PROGRAM Manual_1
VAR
	running: BOOL;
	currentError: UDINT;
	manualMode: E_JogMode;
	velocity: LREAL;
	acceleration: LREAL;
	deceleration: LREAL;
	jerk: LREAL;
	done: BOOL;
	busy: BOOL;
	reset: BOOL;
END_VAR

RAVL.axis.ReadStatus();


RAVL.axisPower(
	Axis:= RAVL.axis,
	Enable:= RAVL.enable,
	Enable_Positive:= RAVL.enable,
	Enable_Negative:= RAVL.enable,
	Override:= RAVL.override,
	BufferMode:= ,
	Options:= ,
	Status=> RAVL.running,
	Busy=> ,
	Active=> ,
	Error=> ,
	ErrorID=> currentError
);

RAVL.axisMoveManual(
	Axis:= RAVL.axis,
	JogForward:= RAVL.forward,
	JogBackwards:= RAVL.backwards,
	Mode:= ,
	Position:= ,
	Velocity:= ,
	Acceleration:= ,
	Deceleration:= ,
	Jerk:= ,
	Done=> RAVL.done,
	Busy=> RAVL.busy,
	Active=> ,
	CommandAborted=> ,
	Error=> ,
	ErrorID=> );

IF RAVL.busy THEN
	RAVL.axisReadActualPosition(Axis := RAVL.axis, Enable := TRUE, Valid=>, Busy=>, Error=>, ErrorID=>, Position=> RAVL.actualPosition);
END_IF
RAVL.actualPositionInt := LREAL_TO_INT(RAVL.actualPosition);

RAVL.axisErrorReset(Axis := RAVL.axis, Execute := RAVL.resetError, Done =>, Error =>, ErrorID => currentError);

END_PROGRAM

(* stored: Version 1.1.0.1, ProductVersion 3.1.4024.6
   POU Manual_1: Id {e5fa7945-e802-46a9-800f-6db9cf40bcd4}, SpecialFunc None *)
